TYPE "Recipe_ShW"
VERSION : 0.1
   STRUCT
      NameFeedBack : String[48];
      "Version" : Int;
      Data1 : Real;
   END_STRUCT;

END_TYPE

